PROGRAM MAIN
VAR
END_VAR

END_PROGRAM

(* stored: Version 1.1.0.1
   POU MAIN: Id {50988f39-9552-4849-95b9-9ffab89a4826} *)
